Staubli VAL3: onF5Event.pgx

program onF5Event()
  local string l_sMessage
  local num l_nActual
  local num l_nOldValue
  local num l_nMoveType
  local num l_nIndex
  local num l_nKey
  local string l_sEvent
begin
end
